TYPE T_Ctrl_SIf_COS_Par :
STRUCT
END_STRUCT
END_TYPE

(* stored: Version 1.1.0.1, ProductVersion 3.1.0.19
   DUT T_Ctrl_SIf_COS_Par: Id {f3e7490b-0041-45c7-8d08-6046729e915c} *)
